{attribute 'qualified_only'}
{attribute 'strict'}
TYPE E_SortingResult :
(
	UNKNOWN				:= 0,
	GOOD 				:= 10,
	CONTAMINATION_DIRTY	:= 20,
	SCRATCH_DENT		:= 30,
	REJECT				:= 40
);
END_TYPE

(* stored: Version 1.1.0.1, ProductVersion 3.1.4024.9
   DUT E_SortingResult: Id {2bc22ade-a5e0-463c-9bd7-ccaed6211ed0} *)
